RoboDK station: SpiralMeca.rdk

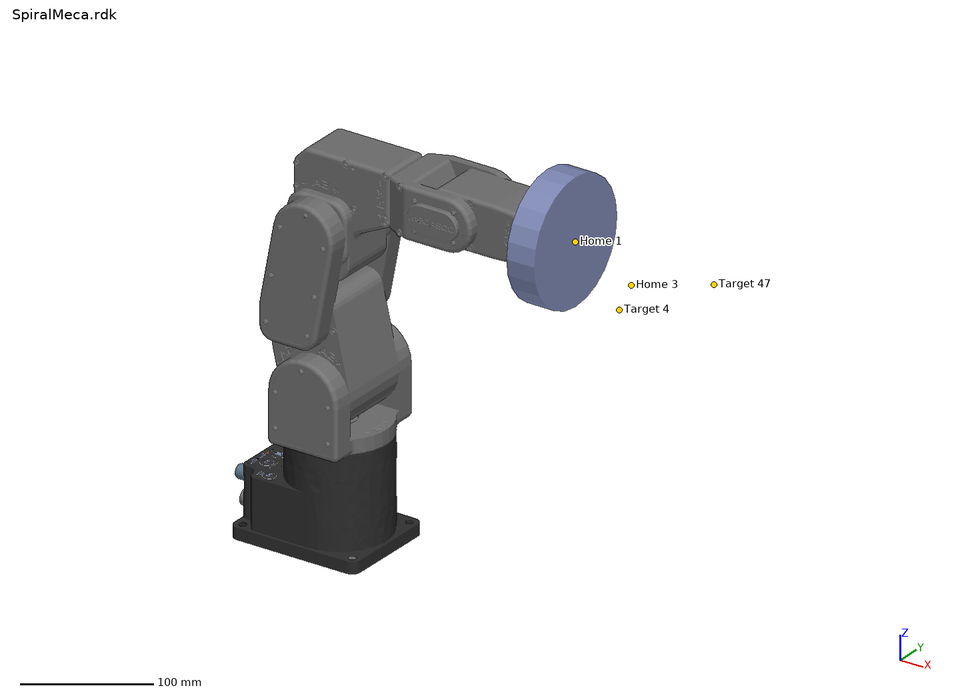
[picture v0: the station drawn from its stored meshes, robots at their saved joint values, targets as dots, program paths as lines]
Station SpiralMeca (saved by RoboDK 5.5.2). Poses are relative to the parent item; angles as X-Y-Z fixed-axis rotations.
  - robot Mecademic Meca500 R3: 6 axes
      modified DH rows (alpha deg, a mm, theta deg, d mm): 0, 0, 0, 135; -90, 0, -90, 0; 0, 135, 0, 0; -90, 38, 0, 120; 90, 0, 0, 0; -90, 0, 180, 70
      joint limits [-150, -70, -135, -170, -115, -720] to [150, 90, 70, 170, 115, 720]; home [0, 0, 0, 0, 0, 0]; saved at [0, 0, 0, 0, 0, 0]
    - tool CrystalToolSample, TCP at (0, 0, 125.4) mm, size 107.9 x 25.4 x 107.9 mm, geometry from CrystalToolSample.STEP
  - frame Frame 1 at (0, 1030, 0) mm
    - target Target 4 (joint target) at (255.71, -1030, 262.52) mm, rotated rx 90 ry -0.21 rz 90 deg; joints [0, -29.636, 42.568, 0, -12.932, 90.212] of Mecademic Meca500 R3
    - target Home 3 (Cartesian target) at (245.4, -1000, 268) mm, rotated rx 0 ry 90 rz 0 deg; joints [0, 10.295, 7.197, 0, -17.492, 0] of Mecademic Meca500 R3
    - target Home 1 (joint target) at (215.4, -1030, 308) mm, rotated rx 0 ry 90 rz 0 deg; joints [0, 0, 0, 0, 0, 0] of Mecademic Meca500 R3
    - target Target 47 (joint target) at (342.4, -1030, 308) mm, rotated rx 0 ry 90 rz 0 deg; joints [0, 11.211, -12.445, 0, 1.234, 0] of Mecademic Meca500 R3
    - target Target 2 (joint target) at (215.4, -1030, 308) mm, rotated rx 0 ry 90 rz 0 deg; joints [0, 0, 0, 0, 0, 0] of Mecademic Meca500 R3
  - Python program Spiral (listed below)
  - Python program Go Home (listed below)
  - Python program SSAP (listed below)
  - Python program Prog4 (listed below)
  - Python program Prog5 (listed below)
  - Python program Prog6 (listed below)
  - Python program Prog7 (listed below)

--- Python program Spiral ---
"""
Created on Thu Jan 19 18:43:18 2023

@author: westj
"""
from robodk.robolink import *       # import the robolink library (bridge with RoboDK)
RDK = Robolink()
from robodk.robomath import *
import math
import numpy as np
import matplotlib.pyplot as plt

class Spiral:
    def __init__(self,x0:float,y0:float,points:float) -> None:
        self.x0=x0 #x offset
        self.y0=y0 #y offset
        self.points=points

    def build(self, radius:float, spacing:float):
        revs=radius/spacing            #calc number of revolutions
        k=spacing/(2*np.pi)
        theta=np.array(np.linspace(0,revs*2*np.pi,self.points)) #how many points and angle coord
        r=k * theta                       #radius coord
        x=(r*np.cos(theta)+self.x0)
        y=(r*np.sin(theta)+self.y0)             #convert to y cartesian

        return x, y #convert to x cartesian


if __name__=="__main__":
    print('Calling spiral from class')
    R=30
    S=10
    TSpeed=10
    cur_spiral=Spiral(0,0,500)
    x,y=cur_spiral.build(R,S)


 #   print(cur_spiral.build(R,S))
  #  plt.plot(x, y, color = 'red', marker = "o")
  #  plt.axis('equal')
  #  plt.show()

#______Robot Movement_________________________________________

robot = RDK.Item('Mecademic Meca500 R3')
home = RDK.Item('Home 1')
target = RDK.Item('Target 2')# retrieve the Target item


robot.MoveJ(home)

robot.MoveJ(target)                 # move the robot to the target
#for i in x:
    #robot.MoveL(target.Pose()*transl(coord))

for i in range(len(x)):

    coord=(x[i],y[i],0)
    robot.MoveJ(target.Pose()*transl(coord))
    robot.WaitFinished()
    #print(coord)
    #print('')

--- Python program Go Home ---
# Type help("robodk.robolink") or help("robodk.robomath") for more information
# Press F5 to run the script
# Documentation: https://robodk.com/doc/en/RoboDK-API.html
# Reference:     https://robodk.com/doc/en/PythonAPI/robodk.html
# Note: It is not required to keep a copy of this file, your Python script is saved with your RDK project

# You can also use the new version of the API:
from robodk import robolink    # RoboDK API
from robodk import robomath    # Robot toolbox
RDK = robolink.Robolink()

robot = RDK.Item('Mecademic Meca500 R3')
home = RDK.Item('Home 1')
robot.MoveJ(home)

--- Python program SSAP ---
"""
Created on Thu Jan 19 18:43:18 2023

@author: westj
"""
from robodk.robolink import *       # import the robolink library (bridge with RoboDK)
RDK = Robolink()
from robodk.robomath import *
import math
import numpy as np
import matplotlib.pyplot as plt
import array
import pandas as pd
from scipy.signal import find_peaks
from scipy.stats import linregress

class Spiral:
    def __init__(self,x0:float,y0:float,points:float) -> None:
        self.x0=x0 #x offset
        self.y0=y0 #y offset
        self.points=points

    def build(self, radius:float, spacing:float):
        revs=radius/spacing            #calc number of revolutions
        k=spacing/(2*np.pi)
        theta=np.array(np.linspace(0,revs*2*np.pi,self.points)) #how many points and angle coord
        r=k * theta                       #radius coord
        x=(r*np.cos(theta)+self.x0)       #convert to x cartesian
        y=(r*np.sin(theta)+self.y0)       #convert to y cartesian

        return x, y

class Linear:
    def __init__(self,data,points):
        self.data=data #data
        self.points=points #x offset

    def get(self,x):
        peaks= find_peaks(self.data['Intensity'], height=.1)

        H=peaks[1]['peak_heights']
        A=[]
        for i in range(len(IPeaks)):
            corr=[IPeaks[i],H[i]]
            A.append(corr)
        SA=sorted(A, key=lambda x: x[1], reverse=True) #sort by peak height largest to smallest
        print(SA)
        XPP=[]
        YPP=[]
        for i in range(self.points):
            #ICP.append(SA[i][0])
            XPP.append(self.data['X'][SA[i][0]])
            YPP.append(self.data['Y'][SA[i][0]])
        LRR=linregress(XPP,YPP)

        return LRR[0]*x+LRR[1]


class Intensity: #intensity function is a gaussian curve
    def __init__(self,x0:float,y0:float, mu_x, mu_y, sigma_x, sigma_y):
        self.x0=-x0 #x offset
        self.y0=-y0 #y offset
        self.mu_x=mu_x
        self.mu_y=mu_y
        self.sigma_x=sigma_x #x squish/stretch
        self.sigma_y=sigma_y #y sqush/stretch


    def get(self,x, y): #gaussian curve definition
        I=np.exp(-0.5 * (((x +self.x0- self.mu_x) / self.sigma_x)**2 + ((y+self.y0 - self.mu_y) / self.sigma_y)**2))
        return I


#*****************************************************************************************************************
#___Initialization______________
xl=0
yl=0
Loops=3
robot = RDK.Item('Mecademic Meca500 R3')
home = RDK.Item('Home 1')
target = RDK.Item('Target 2')# retrieve the Target item

robot.MoveJ(home)
robot.MoveJ(target)



for L in range(1,Loops+1):
    print(L)
    if __name__=="__main__":
        print('Calling spiral from class')

        cur_spiral=Spiral(xl,yl,200) #setting params of the spiral we will be using
        x,y=cur_spiral.build(10/L**L,5/L) #build our spiral x y coords
        Ix=1.24
        Iy=-2.3
        TestInt=Intensity(Ix,Iy,0,0,10,10) #set test intensity parameters

        #Plot our spiral
        # plt.plot(x, y, color = 'red', marker = "o")
        # plt.axis('equal')
        # plt.show()

    #initialize params
    X=[]
    Y=[]
    Z=[]
    Iv=[]
    Cv=[]

    for i in range(len(x)): #loop to get coord and corresponding intensity
        coord=(x[i],y[i],0)
        X.append(x[i])
        Y.append(y[i])
        Z.append(0)
        Ic=TestInt.get(x[i],y[i])
        Iv.append(np.array(Ic))

        robot.MoveJ(target.Pose()*transl(coord))
        robot.WaitFinished()
        #pandas dictionary
        titled_columns={'X': X,'Y': Y,'Z': Z,
                        'Intensity': Iv}
        data = pd.DataFrame(titled_columns)


    peaks= find_peaks(data['Intensity'], height=.1)
    IPeaks=peaks[0]
    H=peaks[1]['peak_heights']
    A=[]
    for i in range(len(IPeaks)):
        corr=[IPeaks[i],H[i]]
        A.append(corr)



    SA=sorted(A, key=lambda x: x[1], reverse=True) #sort by peak height largest to smallest
    if len(SA) == 1:
        print('one peak detected')
        break
    else:

     CL=Linear(data,2) #current linear line definition

    step=.1/L #linear step size
    xl=data['X'][SA[0][0]] #start x
    yl=CL.get(xl) #start y

    Xl=[xl]
    Yl=[yl]
    Il=[TestInt.get(xl,yl)]

    if  data['X'][SA[0][0]] < data['X'][SA[1][0]]:
        step=step
    else:
        step=-step


    while TestInt.get(xl+step,CL.get(xl+step)) >= TestInt.get(xl,CL.get(xl)):

        xl=xl+step
        yl=CL.get(xl)
        il=TestInt.get(xl,yl)
        Xl.append(xl)
        Yl.append(yl)
        Il.append(il)
        coord=(xl,yl,0)
        robot.MoveJ(target.Pose()*transl(coord))



    LLdata={'X':Xl,'Y':Yl,'I':Il}
    Ldata=pd.DataFrame(LLdata)

    fig = plt.figure()
    plt.style.use('seaborn-notebook')
    ax = fig.add_subplot(111, projection='3d')
    ax.plot3D(data['X'], data['Y'], data['Intensity'])
    ax.plot3D(data['X'][IPeaks], data['Y'][IPeaks], data['Intensity'][IPeaks],"x")
    ax.plot3D(Xl, Yl, Il,'o')

    ax.set_xlabel('X axis')
    ax.set_ylabel('Y axis')
    ax.set_zlabel('Z axis')
plt.show()




E=np.sqrt((Ix-xl)**2+(Iy-yl)**2)
print('***Linear Translation********************************************************')
print(Ldata)
print('_________SSAP Report:_________')
print('Calculated peak is at',xl,yl)
print('True peak is at',Ix,Iy)
print('Error is:',E)
print('Linear step size is:',step)

--- Python program Prog4 ---
# -*- coding: utf-8 -*-
"""
Created on Tue Feb 14 10:13:50 2023

@author: ChatGPT/ Jeremy West
"""

import math
from robodk.robolink import *
from robodk import robomath
RDK = Robolink()

target = RDK.Item('Target 2')# retrieve the Target item
robot = RDK.Item('Mecademic Meca500 R3')

# Define the position of the robot's tool
x = 100
y = 100
z = 300

# Define the orientation of the robot's tool using Euler angles (in degrees)
a = 0   # rotation around x-axis
b = 0    # rotation around y-axis
g = 0    # rotation around z-axis


# Set the robot's tool pose to the defined pose
#robodk.robomath.TxyzRxyz_2_Pose(xyzrpw) #[x,y,z,a,b,g]

#pose=robodk.robomath.Pose([x,y,z,a,b,g])
robot.setJoints([0,0,0,0,0,0])
robot.MoveJ(target)
approach = target.Pose()*transl(0,0,-100)
robot.MoveL(approach)

#print(pose)


robot.setPose(pose)

--- Python program Prog5 ---
from robodk.robolink import *       # import the robolink library (bridge with RoboDK)
from robodk.robomath import *       # import the robotics toolbox
RDK = Robolink()                    # establish a link with the simulator
robot = RDK.Item('Mecademic Meca500 R3')     # retrieve the robot by name
robot.setJoints([0,0,0,0,0,0])      # set all robot axes to zero


target = RDK.Item('Target 2')         # retrieve the Target item
robot.MoveJ(target)                 # move the robot to the target

# calculate a new approach position 100 mm along the Z axis of the tool with respect to the target

# Define the position of the robot's tool
x = 255
y = -1030
z = 262

# Define the orientation of the robot's tool using Euler angles (in degrees)
a = 0   # rotation around x-axis
b = 90    # rotation around y-axis
g = 90    # rotation around z-axis

pose=Pose(x,y,z,a,b,g)


approach = target.Pose()*transl(10,-20,0)
print(target.Pose())
robot.MoveL(approach)               # linear move to the approach position

print('approach reached')
print('Attempting pose', pose)
#robot.MoveL(pose)

--- Python program Prog6 ---
# Type help("robodk.robolink") or help("robodk.robomath") for more information
# Press F5 to run the script
# Documentation: https://robodk.com/doc/en/RoboDK-API.html
# Reference:     https://robodk.com/doc/en/PythonAPI/robodk.html
# Note: It is not required to keep a copy of this file, your Python script is saved with your RDK project

# You can also use the new version of the API:
from robodk import robolink    # RoboDK API
from robodk import robomath    # Robot toolbox
RDK = robolink.Robolink()

# Forward and backwards compatible use of the RoboDK API:
# Remove these 2 lines to follow python programming guidelines
from robodk import *      # RoboDK API
from robolink import *    # Robot toolbox
# Link to RoboDK
# RDK = Robolink()

# Notify user:
print('To edit this program:\nright click on the Python program, then, select "Edit Python script"')

# Program example:
item = RDK.Item('base')
if item.Valid():
    print('Item selected: ' + item.Name())
    print('Item posistion: ' + repr(item.Pose()))

print('Items in the station:')
itemlist = RDK.ItemList()
print(itemlist)

# Provoking an exception will display the console output if you run this script from RoboDK
raise Exception('Program not edited.')

--- Python program Prog7 ---
"""
Created on Thu Jan 19 18:43:18 2023

@author: westj
"""
from robodk.robolink import *       # import the robolink library (bridge with RoboDK)
RDK = Robolink()
from robodk.robomath import *
import math
import numpy as np
import matplotlib.pyplot as plt
import array
import pandas as pd
import requests
import re
from scipy.signal import find_peaks
from scipy.stats import linregress

class Spiral:
    def __init__(self,x0:float,y0:float,points:float) -> None:
        self.x0=x0 #x offset
        self.y0=y0 #y offset
        self.points=points

    def build(self, radius:float, spacing:float):
        revs=radius/spacing            #calc number of revolutions
        k=spacing/(2*np.pi)
        theta=np.array(np.linspace(0,revs*2*np.pi,self.points)) #how many points and angle coord
        r=k * theta                       #radius coord
        x=(r*np.cos(theta)+self.x0)       #convert to x cartesian
        y=(r*np.sin(theta)+self.y0)       #convert to y cartesian

        return x, y

class Linear:
    def __init__(self,data,points):
        self.data=data #data
        self.points=points #x offset

    def get(self,x):
        peaks= find_peaks(self.data['Intensity'], height=.1)

        H=peaks[1]['peak_heights']
        A=[]
        for i in range(len(IPeaks)):
            corr=[IPeaks[i],H[i]]
            A.append(corr)
        SA=sorted(A, key=lambda x: x[1], reverse=True) #sort by peak height largest to smallest
        print(SA)
        XPP=[]
        YPP=[]
        for i in range(self.points):
            #ICP.append(SA[i][0])
            XPP.append(self.data['X'][SA[i][0]])
            YPP.append(self.data['Y'][SA[i][0]])
        LRR=linregress(XPP,YPP)

        return LRR[0]*x+LRR[1]


class Intensity: #intensity function is a gaussian curve
    def __init__(self,x0:float,y0:float, mu_x, mu_y, sigma_x, sigma_y):
        self.x0=-x0 #x offset
        self.y0=-y0 #y offset
        self.mu_x=mu_x
        self.mu_y=mu_y
        self.sigma_x=sigma_x #x squish/stretch
        self.sigma_y=sigma_y #y sqush/stretch


    def get(self,x, y): #gaussian curve definition
        I=np.exp(-0.5 * (((x +self.x0- self.mu_x) / self.sigma_x)**2 + ((y+self.y0 - self.mu_y) / self.sigma_y)**2))
        return I

class Photoresistor:
    def __init__(self,url) -> None:
        self.url=url
    def get(self):
        response = requests.get(self.url)
        if response.ok:
            value = response.text
            PR=re.findall(r'\d+',value)
            print('Received value:', value)
            print('Number', PR)
        else:
            print('Error:', response.status_code)
            return -int(PR[0])


#*****************************************************************************************************************
#___Initialization______________
xl=0
yl=0
Loops=3
robot = RDK.Item('Mecademic Meca500 R3')
home = RDK.Item('Home 1')
target = RDK.Item('Target 2')# retrieve the Target item
PR=Photoresistor( 'http://192.168.0.24')

robot.MoveJ(home)
robot.MoveJ(target)



for L in range(1,Loops+1):
    print(L)
    if __name__=="__main__":
        print('Calling spiral from class')

        cur_spiral=Spiral(xl,yl,200) #setting params of the spiral we will be using
        x,y=cur_spiral.build(5/L**L,1/L) #build our spiral x y coords
        Ix=1.24
        Iy=-2.3
        TestInt=Intensity(Ix,Iy,0,0,10,10) #set test intensity parameters

        #Plot our spiral
        # plt.plot(x, y, color = 'red', marker = "o")
        # plt.axis('equal')
        # plt.show()

    #initialize params
    X=[]
    Y=[]
    Z=[]
    Iv=[]
    Cv=[]

    for i in range(len(x)): #loop to get coord and corresponding intensity
        coord=(x[i],y[i],0)
        X.append(x[i])
        Y.append(y[i])
        Z.append(0)
        Ic=PR.get()
        Iv.append(np.array(Ic))

        robot.MoveJ(target.Pose()*transl(coord))
        robot.WaitFinished()
        #pandas dictionary
        titled_columns={'X': X,'Y': Y,'Z': Z,
                        'Intensity': Iv}
        data = pd.DataFrame(titled_columns)


    peaks= find_peaks(data['Intensity'], height=.1)
    IPeaks=peaks[0]
    H=peaks[1]['peak_heights']
    A=[]
    for i in range(len(IPeaks)):
        corr=[IPeaks[i],H[i]]
        A.append(corr)



    SA=sorted(A, key=lambda x: x[1], reverse=True) #sort by peak height largest to smallest
    if len(SA) == 1:
        print('one peak detected')
        break
    else:

     CL=Linear(data,2) #current linear line definition

    step=.1/L #linear step size
    xl=data['X'][SA[0][0]] #start x
    yl=CL.get(xl) #start y

    Xl=[xl]
    Yl=[yl]
    PRS=0
    Il=[0]

    if  data['X'][SA[0][0]] < data['X'][SA[1][0]]:
        step=step
    else:
        step=-step


    while PR.get() >= PRS:

        xl=xl+step
        yl=CL.get(xl)
        PRS=PR.get()
        Xl.append(xl)
        Yl.append(yl)
        Il.append(PRS)
        coord=(xl,yl,0)
        robot.MoveJ(target.Pose()*transl(coord))



    LLdata={'X':Xl,'Y':Yl,'I':Il}
    Ldata=pd.DataFrame(LLdata)

    fig = plt.figure()
    plt.style.use('seaborn-notebook')
    ax = fig.add_subplot(111, projection='3d')
    ax.plot3D(data['X'], data['Y'], data['Intensity'])
    ax.plot3D(data['X'][IPeaks], data['Y'][IPeaks], data['Intensity'][IPeaks],"x")
    ax.plot3D(Xl, Yl, Il,'o')

    ax.set_xlabel('X axis')
    ax.set_ylabel('Y axis')
    ax.set_zlabel('Z axis')
plt.show()




E=np.sqrt((Ix-xl)**2+(Iy-yl)**2)
print('***Linear Translation********************************************************')
print(Ldata)
print('_________SSAP Report:_________')
print('Calculated peak is at',xl,yl)
print('True peak is at',Ix,Iy)
print('Error is:',E)
print('Linear step size is:',step)
